Yaskawa INFORM job: SKRZYNIA_5440_-90_STOPNI_20BR.JBI

/JOB
//NAME SKRZYNIA_5440_-90_STOPNI_20BR
///FOLDERNAME 02-SKRZYNIE_JOBS
//POS
///NPOS 563,563,0,37,0,0
///TOOL 0
///POSTYPE PULSE
///PULSE
C00000=0,-52280,40443,0,6876,0
C00001=-82314,-24956,17040,-59626,-27382,-6248
C00002=-93910,-8625,17040,-59626,-43355,-6248
C00003=-98846,-1061,-42166,-80308,-57081,16120
C00004=-100452,6057,-48127,-85711,-56704,21322
C00005=-95817,31791,-34187,-84788,-63710,26674
C00006=-95573,33077,-33257,-84645,-64023,26851
C00007=-94315,33778,-32137,-85160,-63467,26714
C00008=-95573,33077,-33257,-84645,-64023,26851
C00009=-94948,31301,-36075,-85235,-63717,27152
C00010=-95573,33077,-33257,-84645,-64023,26851
C00011=-95263,33142,-33256,-84677,-63995,26850
C00012=-95263,33142,-33256,-84677,-63995,26850
C00013=-94230,33719,-32331,-85099,-63538,26735
C00014=-95263,33142,-33256,-84677,-63995,26850
C00015=-94794,31816,-35365,-85120,-63763,27076
C00016=-95263,33142,-33256,-84677,-63995,26850
C00017=-95260,33144,-33256,-84678,-63995,26850
C00018=-95260,33144,-33256,-84678,-63995,26850
C00019=-94260,33701,-32361,-85086,-63552,26738
C00020=-95260,33144,-33256,-84678,-63995,26850
C00021=-94835,31943,-35167,-85080,-63786,27056
C00022=-95260,33144,-33256,-84678,-63995,26850
C00023=-95258,25631,32269,-66559,-75499,2416
C00024=-95258,25631,32269,-66559,-75499,2416
C00025=-94256,26435,33444,-66420,-74940,2208
C00026=-95258,25631,32269,-66559,-75499,2416
C00027=-94857,24030,29962,-66606,-75105,2539
C00028=-95258,25631,32269,-66559,-75499,2416
C00029=-98811,21047,-15512,-99242,-81394,20987
C00030=-98811,21047,-15512,-99242,-81394,20987
C00031=-97856,21592,-14760,-99539,-80803,20995
C00032=-98811,21047,-15512,-99242,-81394,20987
C00033=-98487,19855,-17143,-99373,-81250,21110
C00034=-98811,21047,-15512,-99242,-81394,20987
C00035=-99077,36985,67047,-90824,-74996,11
C00036=-99077,36985,67047,-90824,-74996,11
C00037=-98126,38026,68808,-90519,-74354,-175
C00038=-99077,36985,67047,-90824,-74996,11
C00039=-98675,34279,62554,-90994,-74807,523
C00040=-99077,36985,67047,-90824,-74996,11
C00041=-98046,30065,45001,-99674,-75008,5996
C00042=-96663,27244,32711,-106417,-76052,10001
C00043=-96035,27733,33435,-106407,-75606,10011
C00044=-96663,27244,32711,-106417,-76052,10001
C00045=-96274,25568,30264,-106516,-75947,10234
C00046=-96663,27244,32711,-106417,-76052,10001
C00047=-93416,-2088,4699,-99676,-50441,9343
C00048=-88080,-20128,-3199,-80943,-31244,2335
C00049=-48287,-55439,-44481,-48508,-5390,-10469
C00050=-48287,-44591,-17414,-16172,-14532,-25809
C00051=-73855,-32171,-5678,-43952,-33220,-11069
C00052=-84843,-2315,38096,-46044,-43440,-11681
C00053=-99590,25338,21334,-81459,-78469,-3358
C00054=-99590,25338,21334,-81459,-78469,-3358
C00055=-98681,25943,22203,-81468,-77867,-3455
C00056=-99590,25338,21334,-81459,-78469,-3358
C00057=-99296,24016,19444,-81525,-78239,-3225
C00058=-99590,25338,21334,-81459,-78469,-3358
C00059=-99820,26032,21623,-82067,-78848,-4447
C00060=-99820,26032,21623,-82067,-78848,-4447
C00061=-98898,26645,22513,-82083,-78237,-4546
C00062=-99820,26032,21623,-82067,-78848,-4447
C00063=-99438,24292,19129,-82156,-78552,-4268
C00064=-99820,26032,21623,-82067,-78848,-4447
C00065=-95331,1432,-9864,-84798,-60031,-3557
C00066=-91210,-11403,-27677,-113165,-52408,5733
C00067=-98271,-15326,-41207,-114268,-59488,7673
C00068=-83743,-25164,-57719,-138536,-50905,17366
C00069=-83743,-25361,-52011,-136459,-47698,15842
C00070=-93071,-30029,-62286,-132724,-54351,14554
C00071=-61872,-66272,-83954,-148251,-32298,21081
C00072=-61872,-49557,-32264,-110357,-15428,1928
C00073=-65143,-26385,24751,-20080,-56896,-30933
C00074=-90244,4395,51028,-38516,-59607,-23032
C00075=-79356,-9150,9683,-42499,-40407,-18801
C00076=-98951,25836,42573,-74290,-75705,-4216
C00077=-99097,30513,38864,-76423,-80199,-875
C00078=-97872,31473,40332,-76298,-79437,-1085
C00079=-99097,30513,38864,-76423,-80199,-875
C00080=-98774,28880,36400,-76469,-79893,-679
C00081=-99097,30513,38864,-76423,-80199,-875
C00082=-99862,24525,29609,-86160,-76987,1407
C00083=-99452,22245,7122,-97683,-80070,9369
C00084=-99292,23987,9562,-97373,-81102,9104
C00085=-98184,24694,10564,-97522,-80343,9095
C00086=-99292,23987,9562,-97373,-81102,9104
C00087=-99030,22873,7999,-97442,-80972,9229
C00088=-99292,23987,9562,-97373,-81102,9104
C00089=-95017,-9844,-333,-79976,-47193,-2364
C00090=-62804,-32782,1918,-36164,-30925,-23493
C00091=-48283,-21883,28214,-25170,-26491,48363
C00092=-45951,-10962,51022,-17493,-32991,44756
C00093=-50347,-18571,12268,-49104,-16423,60029
C00094=-52008,-16476,13921,-52720,-16985,61589
C00095=-50839,-15356,14836,-51561,-16264,61168
C00096=-51137,-15647,14596,-51864,-16447,61279
C00097=-52695,-14846,15261,-54465,-17168,62360
C00098=-51384,-16746,13703,-51673,-16698,61154
C00099=-50347,-18571,12268,-49104,-16423,60029
C00100=-52476,-17044,12146,-55476,-16783,62883
C00101=-51467,-16091,12918,-54586,-16145,62570
C00102=-51762,-16375,12685,-54854,-16332,62665
C00103=-53129,-15664,13268,-57063,-16995,63582
C00104=-52557,-17119,12084,-55547,-16837,62908
C00105=-50509,-19000,10610,-51503,-15997,61182
C00106=-52966,-16930,12240,-56194,-17032,63176
C00107=-51879,-15912,13067,-55265,-16346,62852
C00108=-52154,-16175,12851,-55507,-16521,62938
C00109=-53227,-15612,13314,-57215,-17042,63646
C00110=-52966,-16930,12240,-56194,-17032,63176
C00111=-50703,-18403,11066,-52155,-16024,61477
C00112=-52780,-17619,11680,-55562,-17015,62889
C00113=-51306,-16241,12790,-54268,-16084,62435
C00114=-51660,-16583,12512,-54593,-16308,62551
C00115=-53327,-15718,13220,-57282,-17114,63667
C00116=-52780,-17619,11680,-55562,-17015,62889
C00117=-50704,-18401,11069,-52157,-16021,61478
C00118=-53191,-17342,11901,-56260,-17204,63181
C00119=-51773,-16022,12969,-55050,-16305,62760
C00120=-52146,-16378,12679,-55379,-16540,62876
C00121=-53214,-15820,13135,-57085,-17059,63584
C00122=-53002,-17172,12037,-56105,-17083,63128
C00123=-51005,-17995,11387,-52847,-16122,61778
C00124=-52654,-17319,11922,-55560,-16911,62904
C00125=-51372,-16113,12897,-54432,-16099,62508
C00126=-51648,-16379,12679,-54684,-16273,62598
C00127=-52952,-15703,13233,-56807,-16903,63480
C00128=-53323,-17134,12070,-56539,-17248,63304
C00129=-52826,-20105,4812,-63938,-15678,66983
C00130=-52298,-19620,5183,-63681,-15322,66914
C00131=-51076,-18450,6096,-63049,-14499,66733
C00132=-51419,-18785,5831,-63233,-14731,66786
C00133=-52680,-18133,6347,-65138,-15424,67581
C00134=-52924,-19431,7025,-60935,-16175,65505
C00135=-51752,-18759,10786,-53484,-16613,62002
C00136=-52244,-17884,11471,-54682,-16766,62529
C00137=-50303,-16031,12961,-52880,-15542,61887
C00138=-50741,-16464,12607,-53310,-15818,62044
C00139=-52416,-15612,13306,-56135,-16617,63223
C00140=-51898,-18011,11369,-54129,-16600,62301
C00141=-50945,-18019,11363,-52741,-16103,61737
C00142=-51347,-17395,11856,-53690,-16237,62152
C00143=-49990,-16073,12923,-52376,-15383,61677
C00144=-50384,-16465,12603,-52769,-15629,61822
C00145=-52066,-15616,13298,-55654,-16423,63028
C00146=-51792,-17610,11685,-54205,-16494,62350
C00147=-50945,-18019,11363,-52741,-16103,61737
C00148=-50845,-17493,11778,-52895,-15987,61824
C00149=-49521,-16191,12826,-51571,-15155,61341
C00150=-49894,-16567,12520,-51958,-15389,61484
C00151=-51728,-15654,13268,-55171,-16246,62832
C00152=-51082,-17431,11827,-53280,-16102,61986
C00153=-50028,-23690,-6096,-22921,-31075,54538
C00154=-50346,-22995,-5584,-23393,-31002,54768
C00155=-48843,-21430,-4410,-21901,-30270,54078
C00156=-49178,-21788,-4683,-22239,-30433,54235
C00157=-50538,-21100,-4158,-23908,-30654,55032
C00158=-50252,-22811,-5450,-23315,-30936,54734
C00159=-49763,-24818,-32918,-23163,-28604,59699
C00160=-49144,-24298,-32242,-22455,-28505,59304
C00161=-47766,-22458,-30816,-21237,-27774,58615
C00162=-48099,-22913,-31171,-21534,-27949,58786
C00163=-49602,-21997,-30448,-23301,-28174,59772
C00164=-49259,-23869,-32392,-22880,-28141,59533
C00165=-50713,-12366,-58367,-41124,-17813,74400
C00166=-50097,-11438,-57505,-40749,-17495,74109
C00167=-49105,-9842,-55994,-40096,-16991,73614
C00168=-49355,-10250,-56383,-40269,-17116,73742
C00169=-50506,-9357,-55529,-41571,-17503,74586
C00170=-49771,-10920,-57018,-40545,-17327,73951
C00171=-46548,-30139,-39639,-20061,-27197,57955
C00172=-48797,-26670,-6576,-20404,-32539,53259
C00173=-45389,-28224,4312,-35967,-15579,54278
C00174=-40154,-51179,-915,-24203,-8234,36524
C00175=0,-52280,40443,0,6876,0
C00176=-2117,-50103,-33543,-4117,45077,85249
C00177=26439,-48928,-33543,-4117,-52362,85249
C00178=26439,-27355,-33543,-41485,-52362,85249
C00179=39218,-24492,-41653,-51934,-39374,86964
C00180=38244,-2284,-24157,-56964,-37300,90090
C00181=26640,586,-20198,-77712,-51919,89712
C00182=26323,460,-20341,-77681,-52125,89737
C00183=25607,3186,-17293,-77585,-52601,89760
C00184=26323,460,-20341,-77681,-52125,89737
C00185=27719,1044,-19697,-77798,-51218,89644
C00186=26640,586,-20198,-77712,-51919,89712
C00187=46457,7101,-11330,-26648,-40775,82885
C00188=47439,8350,-9833,-26106,-40556,82449
C00189=46334,10684,-6981,-26557,-41070,82837
C00190=47439,8350,-9833,-26106,-40556,82449
C00191=48354,9159,-8854,-25603,-40343,82046
C00192=47439,8350,-9833,-26106,-40556,82449
C00193=24760,-3019,-10726,-94610,-54398,89614
C00194=25145,-1220,-8811,-94681,-54143,89655
C00195=24492,1290,-6066,-94601,-54582,89624
C00196=25145,-1220,-8811,-94681,-54143,89655
C00197=26584,-669,-8211,-94866,-53174,89734
C00198=25145,-1220,-8811,-94681,-54143,89655
C00199=14532,-15164,-22494,-92943,-61192,88617
C00200=-33377,-12679,-20251,-90012,-93751,87621
C00201=-32674,-7309,22058,-70557,-98373,80594
C00202=20046,-29908,-41690,-58842,-55822,75080
C00203=46158,10269,-6164,-23128,-46470,70172
C00204=51306,10256,-19432,-23475,-33025,71236
C00205=50386,12004,-17260,-23922,-33430,71616
C00206=51306,10256,-19432,-23475,-33025,71236
C00207=51995,10928,-18601,-23012,-32906,70879
C00208=51306,10256,-19432,-23475,-33025,71236
C00209=50667,8104,-22050,-23976,-33027,71608
C00210=27434,3323,14960,-56922,-57501,78346
C00211=29014,6574,18756,-56344,-56678,77965
C00212=28326,9009,21700,-56459,-57175,78009
C00213=29014,6574,18756,-56344,-56678,77965
C00214=30292,7183,19486,-55908,-55969,77693
C00215=29014,6574,18756,-56344,-56678,77965
C00216=24457,-1296,-8898,-94600,-54606,89622
C00217=24457,-1296,-8898,-94600,-54606,89622
C00218=23939,748,-6672,-94541,-54956,89598
C00219=24457,-1296,-8898,-94600,-54606,89622
C00220=25626,-864,-8432,-94748,-53818,89684
C00221=24457,-1296,-8898,-94600,-54606,89622
C00222=22058,-20035,-26567,-93333,-56013,88551
C00223=-28907,-25632,-31027,-90338,-90583,86609
C00224=-23923,-11573,-19230,-90501,-87328,87840
C00225=-8646,-8251,-7782,-76032,-82054,83740
C00226=42001,26537,64712,-25019,-74648,68382
C00227=42692,25604,59505,-25067,-71864,68798
C00228=42100,27723,62792,-25233,-72628,68820
C00229=42692,25604,59505,-25067,-71864,68798
C00230=43179,26157,60355,-24838,-71882,68629
C00231=42692,25604,59505,-25067,-71864,68798
C00232=42064,17796,48100,-25604,-70267,69397
C00233=28113,-7386,-15136,-95790,-47335,90009
C00234=28228,-6488,-14240,-95859,-47266,90053
C00235=27767,-5044,-12775,-95858,-47588,90072
C00236=28228,-6488,-14240,-95859,-47266,90053
C00237=29468,-5989,-13737,-96077,-46438,90154
C00238=28228,-6488,-14240,-95859,-47266,90053
C00239=51937,664,-7429,-160484,-50080,89770
C00240=52345,1107,-6938,-160727,-50007,89930
C00241=51359,2767,-5080,-160136,-50147,89540
C00242=52345,1107,-6938,-160727,-50007,89930
C00243=53054,1752,-6222,-161147,-49882,90209
C00244=52345,1107,-6938,-160727,-50007,89930
C00245=51937,664,-7429,-160484,-50080,89770
C00246=29691,-10745,-18393,-95770,-46230,89933
C00247=26663,-19279,-25970,-94307,-48104,89008
C00248=29542,-7588,-14846,-100915,-46930,90773
C00249=29616,-6902,-10165,-96183,-45225,84004
C00250=29097,-5391,-8640,-96201,-45588,84023
C00251=29616,-6902,-10165,-96183,-45225,84004
C00252=31098,-6282,-9543,-96410,-44233,84135
C00253=29616,-6902,-10165,-96183,-45225,84004
C00254=7576,-30273,-44451,-97512,-61182,86443
C00255=-18624,-40022,-50597,-93591,-78329,83668
C00256=-32134,-30783,-37092,-96173,-88064,83581
C00257=23774,-1324,-8929,-94512,-55065,89585
C00258=23774,-1324,-8929,-94512,-55065,89585
C00259=23319,517,-6924,-94461,-55372,89567
C00260=23774,-1324,-8929,-94512,-55065,89585
C00261=25077,-853,-8421,-94674,-54188,89653
C00262=23774,-1324,-8929,-94512,-55065,89585
C00263=22107,-1052,28039,-94807,-51389,77849
C00264=19995,-16885,24938,-75612,-39910,62837
C00265=8393,-42921,36369,-24238,-5473,19544
C00266=0,-52280,40443,0,6876,0
C00267=-82314,-24956,17040,-59626,-27382,-6248
C00268=-93910,-8625,17040,-59626,-43355,-6248
C00269=-98846,-1061,-42166,-80308,-57081,16120
C00270=-100452,6057,-48127,-85711,-56704,21322
C00271=-95564,34698,-34234,-85516,-63941,27819
C00272=-94021,36658,-30981,-84167,-64832,27454
C00273=-93851,36773,-30815,-84181,-64812,27439
C00274=-95564,34698,-34234,-85516,-63941,27819
C00275=-96930,32282,-32252,-82595,-65816,26305
C00276=-93901,32995,-31122,-83953,-64436,26132
C00277=-93891,32978,-31150,-83961,-64431,26134
C00278=-96930,32282,-32252,-82595,-65816,26305
C00279=-97719,-4194,-31542,-76086,-54596,10626
C00280=-88377,-34186,-45291,-67238,-52212,2442
C00281=-73560,-62084,7826,-28695,-34737,-3666
C00282=0,-52280,40443,0,6876,0
C00283=0,-52280,40443,0,6876,0
C00284=-2117,-50103,-33543,-4117,45077,85249
C00285=26439,-48928,-33543,-4117,-52362,85249
C00286=26439,-27355,-33543,-41485,-52362,85249
C00287=39218,-24492,-41653,-51934,-39374,86964
C00288=37381,-5106,-22608,-53943,-39515,88347
C00289=38119,-10689,-19379,-70548,-34101,88029
C00290=37906,-14512,-22901,-69984,-34376,87713
C00291=41414,6981,-5927,-33889,-45598,86373
C00292=42289,10624,-1511,-33365,-45508,85956
C00293=42351,10656,-1473,-33340,-45486,85935
C00294=41414,6981,-5927,-33889,-45598,86373
C00295=53221,-12364,-8957,-19277,-47766,73858
C00296=11365,-15171,10010,-30164,-77975,82960
C00297=16156,-38280,11293,-23671,-42998,42040
C00298=11365,-47379,10010,-30164,3063,681
C00299=0,-52280,40443,0,6876,0
C00300=0,-36700,24612,42871,-31823,33862
C00301=-44403,-30110,7154,-24155,-23805,45557
C00302=-51570,-19542,10947,-41619,-21811,53396
C00303=-51570,-17239,16856,-38066,-23574,51584
C00304=-55052,-13712,19754,-43494,-24529,53873
C00305=-55190,-12778,21730,-42693,-25060,53437
C00306=-40431,-28773,9158,-17648,-23273,42875
C00307=0,-36700,24612,42871,-31823,33862
C00308=0,-52280,40443,0,6876,0
C00309=0,-52280,40443,0,6876,0
C00310=-73560,-62084,7826,-28695,-34737,-3666
C00311=-88377,-34186,-45291,-67238,-52212,2442
C00312=-99860,-8392,-35780,-75647,-56000,10650
C00313=-100432,21324,12575,-83706,-77956,7498
C00314=-100432,21324,12575,-83706,-77956,7498
C00315=-97477,24790,17443,-83584,-77881,7143
C00316=-97548,25214,18044,-83537,-78171,7107
C00317=-100432,21324,12575,-83706,-77956,7498
C00318=-100473,21504,12824,-83696,-77986,7482
C00319=-97708,25565,18549,-83502,-78342,7077
C00320=-97720,26100,19317,-83456,-78605,7025
C00321=-100432,21324,12575,-83706,-77956,7498
C00322=-98403,3681,-8965,-86029,-63956,7946
C00323=-98851,2841,7216,-80537,-62817,1838
C00324=-99868,-33,22146,-72719,-59601,-5126
C00325=-99028,-10516,17309,-71061,-60695,-4227
C00326=-58820,-39124,10926,-53325,-41870,-3759
C00327=0,-52280,40443,0,6876,0
C00328=-37281,-50778,-9546,-79570,-75313,71156
C00329=-21038,-23698,-30323,-82948,-81132,85647
C00330=-21230,-24252,-33397,-84866,-81311,86227
C00331=26224,-11477,-22521,-89106,-49066,87170
C00332=30473,789,4724,-68168,-47848,79016
C00333=30460,-1091,-3608,-71823,-46530,81583
C00334=26224,-11477,-22521,-89106,-49066,87170
C00335=1250,-26379,-34995,-85812,-66036,85728
C00336=-29373,-17697,-13794,-84248,-87305,82376
C00337=-12562,-22815,-22029,-52123,-75138,85349
C00338=41964,2536,-13642,-34848,-42769,74522
C00339=37974,4101,-26304,-58477,-36842,84551
C00340=37992,4823,-31618,-63468,-34913,87461
C00341=41439,5489,-14791,-37032,-40569,75962
C00342=38833,-3286,10682,-41231,-51577,69207
C00343=-9276,-22918,-17698,-90837,-69000,78700
C00344=-8172,-56778,-49528,-75726,-40055,75711
C00345=-3982,-61001,-53003,-69042,-33087,73336
C00346=37287,-55159,35520,-2191,5667,2084
C00347=0,-52280,40443,0,6876,0
C00348=0,-36700,24612,42871,-31823,33862
C00349=-44403,-30110,7154,-24155,-23805,45557
C00350=-44403,-30110,7154,-24155,-23805,45557
C00351=-42101,-12213,25656,-103795,-5192,78630
C00352=-46259,-8171,27719,-110365,-8144,81138
C00353=-67532,2461,52564,-58221,-38014,54436
C00354=-67092,2390,52438,-57975,-37749,54380
C00355=-61198,-4613,8805,-137219,-40022,88160
C00356=-56934,-15752,2926,-132390,-27589,90381
C00357=-47073,-34549,9488,-27883,-30316,51458
C00358=0,-52280,40443,0,6876,0
C00359=0,-52280,40443,0,6876,0
C00360=-73560,-62084,7826,-28695,-34737,-3666
C00361=-96366,-17217,16860,-56620,-71703,-18245
C00362=-98152,-14905,2044,-65675,-67485,-3494
C00363=-100467,-7393,-15195,-81625,-60158,6002
C00364=-99336,18440,8642,-84276,-74234,7647
C00365=-99336,18440,8642,-84276,-74234,7647
C00366=-97907,25479,18429,-83510,-78268,7080
C00367=-97774,25771,18838,-83486,-78362,7054
C00368=-99336,18440,8642,-84276,-74234,7647
C00369=-99336,20364,19482,-82786,-74642,4774
C00370=-98337,25059,18813,-87846,-78771,10707
C00371=-98337,23926,10585,-88652,-78855,12971
C00372=-99528,19847,13673,-83665,-74506,6500
C00373=-89817,-17341,-38408,-97132,-45323,12250
C00374=-100347,-21961,-42251,-93939,-52125,11121
C00375=-60204,-59872,-73451,-117647,-17639,18840
C00376=-37721,-67612,11381,-1325,-438,-7850
C00377=0,-52280,40443,0,6876,0
C00378=37287,-55159,35520,-2191,5667,2084
C00379=40042,-68802,-18337,-47708,-19461,45384
C00380=16481,-63411,-38742,-86271,-37962,67106
C00381=28646,-23138,-32952,-89786,-42552,85395
C00382=38882,-16596,-17625,-44304,-41043,72768
C00383=40930,-6862,-13364,-47045,-37020,74415
C00384=41744,-3361,-9781,-46774,-36492,74231
C00385=41678,-4243,-16493,-50979,-33997,76666
C00386=40930,-6862,-13364,-47045,-37020,74415
C00387=38882,-16596,-17625,-44304,-41043,72768
C00388=28646,-23138,-32952,-89786,-42552,85395
C00389=29905,-15291,-26411,-91102,-43435,86304
C00390=31540,-7654,-19248,-92177,-42391,86919
C00391=31445,-8095,-22888,-97196,-43117,89457
C00392=29637,-16450,-35189,-96198,-44206,89682
C00393=-7164,-46429,-55577,-86274,-68578,84143
C00394=40042,-68802,-18337,-47708,-19461,45384
C00395=37287,-55159,35520,-2191,5667,2084
C00396=0,-52280,40443,0,6876,0
C00397=-37164,-60659,6466,-13301,-5027,19773
C00398=-45362,-39990,2831,-27538,-17767,40935
C00399=-57189,-26834,-7130,-38780,-31731,51561
C00400=-55974,-20661,-3180,-39617,-29741,52134
C00401=-55991,-28453,-45977,-64163,-20900,63765
C00402=-57189,-26834,-7130,-38780,-31731,51561
C00403=-41180,-61187,4729,-17280,-8498,23442
C00404=0,-52280,40443,0,6876,0
C00405=0,-52280,40443,0,6876,0
C00406=-43180,-50572,-20637,-6552,-29302,-38834
C00407=-79425,-37128,-15462,-51820,-35721,-18807
C00408=-93702,-21743,-5664,-65079,-41536,-12324
C00409=-94876,-11469,-23586,-124528,-59237,5423
C00410=-92861,23404,17376,-116518,-76732,-1573
C00411=-96665,29896,42633,-98437,-75635,-11031
C00412=-96665,37701,65506,-96077,-73868,-15674
C00413=-98256,26642,30161,-104402,-77650,-7294
C00414=-94876,-11469,-23586,-124528,-59237,5423
C00415=-94108,-26192,-19530,-80749,-38523,-6311
C00416=-79425,-37128,-15462,-51820,-35721,-18807
C00417=-44920,-50063,-20090,-8739,-29356,-37564
C00418=-37721,-67612,11381,-1325,-438,-7850
C00419=0,-52280,40443,0,6876,0
C00420=40043,-68802,-18337,-47706,-19461,45383
C00421=27078,-46675,7729,-35821,-60236,53359
C00422=37661,6027,34279,-36092,-58837,68690
C00423=38848,9668,32452,-36978,-55195,69693
C00424=45203,15557,41040,-24527,-60177,66840
C00425=37661,2340,23735,-37788,-55306,70200
C00426=22173,-30639,7984,-58136,-45615,60133
C00427=37287,-55159,35520,-2191,5667,2084
C00428=0,-52280,40443,0,6876,0
C00429=-23708,-46776,23536,-16027,-4787,19738
C00430=-50917,-40459,4132,-34421,-18173,42391
C00431=-54964,-26842,8528,-44141,-23181,52038
C00432=-51719,-20944,8196,-48593,-18539,54728
C00433=-53338,-16066,12564,-52314,-18938,56375
C00434=-53668,-14237,17353,-48629,-20286,54493
C00435=-18010,-41727,-5437,24633,-20435,23511
C00436=-18010,-41727,-5437,24633,-20435,23511
C00437=-43180,-50572,-20637,-6552,-29302,-38834
C00438=-37721,-67612,11381,-1325,-438,-7850
C00439=0,-52280,40443,0,6876,0
C00440=-7830,-25136,17099,-55306,-64068,52084
C00441=34592,-23156,18291,-29932,-45204,43222
C00442=27626,-5609,7480,-74303,-46810,69713
C00443=30162,-7263,-3756,-79871,-43922,73611
C00444=30945,-3557,12,-79972,-43367,73694
C00445=30934,-3652,-86,-79966,-43372,73693
C00446=29106,-7674,-4162,-79972,-44640,73655
C00447=-2837,-32019,-23857,-80741,-66785,72567
C00448=9534,-43450,13514,-26959,-29486,38723
C00449=22834,-59963,22946,-6692,-2150,9612
C00450=0,-52280,40443,0,6876,0
C00451=-23708,-46776,23536,-16027,-4787,19738
C00452=-50917,-40459,4132,-34421,-18173,42391
C00453=-51059,-36587,4608,-36647,-19418,45358
C00454=-50113,-22729,10834,-36393,-23396,50963
C00455=-58003,-17258,7975,-66354,-22196,69294
C00456=-57660,-15851,11780,-61832,-22634,66694
C00457=-50113,-22729,10834,-36393,-23396,50963
C00458=-45969,-44671,-42317,80322,10570,10889
C00459=-31285,-69981,-10849,-7246,-6842,20992
C00460=0,-52280,40443,0,6876,0
C00461=-37721,-67612,11381,-1325,-438,-7850
C00462=-43180,-50572,-20637,-6552,-29302,-38834
C00463=-92181,-6909,34626,-50562,-49190,-21840
C00464=-101117,-5694,-18308,-85789,-60825,2377
C00465=-97622,-3602,-16155,-86160,-58465,2400
C00466=-99754,24347,18348,-83049,-78046,1543
C00467=-98401,23935,17754,-83131,-77323,1564
C00468=-98274,24050,17917,-83129,-77329,1551
C00469=-99954,24418,19993,-82828,-78557,1051
C00470=-99712,24798,18984,-83012,-78332,1506
C00471=-99852,25442,19906,-82977,-78439,1439
C00472=-98294,26390,21274,-82926,-78604,1336
C00473=-98320,27540,23370,-82787,-79202,1083
C00474=-99852,25442,19906,-82977,-78439,1439
C00475=-99768,8894,-2445,-89351,-68751,3793
C00476=-96099,-3787,-16815,-92200,-58195,4535
C00477=-97559,-25159,-36085,-93407,-46496,3918
C00478=-68601,-52593,-52127,-95725,-25602,3235
C00479=-80632,-38079,-20908,-64053,-45216,-12949
C00480=-43180,-50572,-20637,-6552,-29302,-38834
C00481=-37721,-67612,11381,-1325,-438,-7850
C00482=54026,-30203,28811,7745,-28969,5087
C00483=55906,-29650,27841,6704,-28568,42061
C00484=3910,-49110,-20873,-64325,-51391,71742
C00485=9596,-41005,-15480,-61992,-50741,70573
C00486=34629,-5327,8260,-51720,-47880,65426
C00487=35679,2837,17551,-51053,-47466,65038
C00488=35689,-56,7549,-54586,-44718,67469
C00489=34629,-5327,8260,-51720,-47880,65426
C00490=9596,-41005,-15480,-61992,-50741,70573
C00491=29660,-4584,-26917,-122917,-59269,85605
C00492=30458,-1431,-23593,-123278,-58903,85810
C00493=32051,-581,-21149,-126899,-58917,85995
C00494=28378,-5181,-30467,-124970,-61925,86269
C00495=9596,-41005,-15480,-61992,-50741,70573
C00496=4124,-42500,-16101,-63937,-54198,71061
C00497=22834,-59963,22946,-6692,-2150,9612
C00498=0,-52280,40443,0,6876,0
C00499=-44101,-76445,-48847,-15697,-17168,40457
C00500=-48984,-30078,-36716,-21434,-29637,58750
C00501=-50484,-13386,-55713,-36158,-19724,71897
C00502=-50319,-9878,-52358,-36554,-19395,72071
C00503=-57778,15231,-57159,-77377,-21293,89265
C00504=-57778,15231,-57159,-77377,-21293,89265
C00505=-50484,-13386,-55713,-36158,-19724,71897
C00506=-49763,-25421,-36239,-24565,-26935,60445
C00507=-50529,-22709,-3778,-22940,-31995,54502
C00508=-45389,-28224,4312,-35967,-15579,54278
C00509=-40154,-51179,-915,-24203,-8234,36524
C00510=0,-52280,40443,0,6876,0
C00511=0,-52280,40443,0,6876,0
C00512=-37721,-67612,11381,-1325,-438,-7850
C00513=-43180,-50572,-20637,-6552,-29302,-38834
C00514=-43180,-50572,-20637,-6552,-29302,-38834
C00515=-91233,-13472,9135,-57436,-42793,-15671
C00516=-94453,18451,26397,-64403,-69695,-4898
C00517=-94848,25710,19994,-67599,-74328,1083
C00518=-94734,25454,19627,-67614,-74234,1097
C00519=-94605,24228,10738,-68938,-72404,3439
C00520=-96555,21614,11724,-68276,-72695,2131
C00521=-99000,22482,23037,-75261,-76004,639
C00522=-97210,28604,31066,-74659,-78513,378
C00523=-97154,26647,21384,-75593,-77346,2770
C00524=-100531,16612,13557,-75306,-72509,1088
C00525=-98914,15791,22093,-91892,-69242,2220
C00526=-98524,31242,37673,-92432,-80087,2200
C00527=-98508,35203,51300,-91477,-79539,-794
C00528=-99299,29399,42249,-91532,-77608,155
C00529=-99299,39874,71997,-89061,-76925,-5800
C00530=-98153,38420,66100,-91432,-76531,-4068
C00531=-98147,36464,60868,-91873,-76694,-3060
C00532=-99718,12303,6039,-96207,-71156,6635
C00533=-93032,-8711,-3060,-81304,-48072,-4095
C00534=-98228,-14972,-11291,-81392,-49231,-4002
C00535=-91129,-17870,8831,-66292,-48444,-14183
C00536=-68865,-35989,-5252,-49829,-38105,-21179
C00537=-15566,-52364,-9989,12732,-35649,-46896
C00538=0,-52278,40443,-31822,-65283,46097
C00539=7820,3000,44222,-77356,-66876,70486
C00540=23103,22769,71034,-65639,-61603,67373
C00541=25078,30713,84198,-63240,-61811,65668
C00542=25008,30264,83410,-63369,-61766,65773
C00543=23103,22769,71034,-65639,-61603,67373
C00544=23103,22769,71034,-65639,-61603,67373
C00545=25078,30713,84198,-63240,-61811,65668
C00546=25008,30264,83410,-63369,-61766,65773
C00547=23103,22769,71034,-65639,-61603,67373
C00548=-3014,-20441,-7349,-104591,-68614,79454
C00549=-3014,-20441,-7349,-104591,-68614,79454
C00550=-13238,-21720,-1359,-93359,-59492,72612
C00551=10261,-46634,14475,-36899,-22136,31570
C00552=22834,-59963,22946,-6692,-2150,9612
C00553=0,-52280,40443,0,6876,0
C00554=-23708,-46776,23536,-16027,-4787,19738
C00555=-50917,-40459,4132,-34421,-18173,42391
C00556=-49876,-21948,7530,-68838,-10324,59148
C00557=-46721,-18942,9765,-68167,-8197,59205
C00558=-47734,-15041,12007,-78406,-8476,63945
C00559=-48173,-14749,12492,-78097,-8776,63748
C00560=-42573,-24036,4541,-56448,-5917,54155
C00561=-31287,-69981,-10850,-7253,-6843,20996
C00562=0,-52280,40443,0,6876,0
BC00000=455888
BC00001=445130
BC00002=445130
BC00003=445130
BC00004=445130
BC00005=467179
BC00006=468227
BC00007=468227
BC00008=468227
BC00009=468227
BC00010=468227
BC00011=514421
BC00012=514421
BC00013=514421
BC00014=514421
BC00015=514421
BC00016=514421
BC00017=560588
BC00018=560588
BC00019=560588
BC00020=560588
BC00021=560588
BC00022=560588
BC00023=536404
BC00024=536404
BC00025=536404
BC00026=536404
BC00027=536404
BC00028=536404
BC00029=582458
BC00030=582458
BC00031=582458
BC00032=582458
BC00033=582458
BC00034=582458
BC00035=581206
BC00036=581206
BC00037=581206
BC00038=581206
BC00039=581206
BC00040=581206
BC00041=608443
BC00042=626741
BC00043=626741
BC00044=626741
BC00045=626741
BC00046=626741
BC00047=604255
BC00048=604255
BC00049=627238
BC00050=699121
BC00051=730161
BC00052=730161
BC00053=820815
BC00054=820815
BC00055=820815
BC00056=820815
BC00057=820815
BC00058=820815
BC00059=866263
BC00060=866263
BC00061=866263
BC00062=866263
BC00063=866263
BC00064=866263
BC00065=866263
BC00066=872244
BC00067=872244
BC00068=872244
BC00069=872244
BC00070=872244
BC00071=872244
BC00072=872244
BC00073=967932
BC00074=965893
BC00075=970341
BC00076=974685
BC00077=981233
BC00078=981233
BC00079=981233
BC00080=981233
BC00081=981233
BC00082=979269
BC00083=1044956
BC00084=1044956
BC00085=1044956
BC00086=1044956
BC00087=1044956
BC00088=1044956
BC00089=978491
BC00090=968330
BC00091=919701
BC00092=943157
BC00093=1012084
BC00094=1012084
BC00095=1012084
BC00096=1012084
BC00097=1012084
BC00098=1012084
BC00099=949003
BC00100=953382
BC00101=953382
BC00102=953382
BC00103=953382
BC00104=953382
BC00105=888056
BC00106=888056
BC00107=888056
BC00108=888056
BC00109=888056
BC00110=888056
BC00111=830714
BC00112=830714
BC00113=830714
BC00114=830714
BC00115=830714
BC00116=830714
BC00117=764829
BC00118=764829
BC00119=764829
BC00120=764829
BC00121=764829
BC00122=764829
BC00123=707174
BC00124=707174
BC00125=707174
BC00126=707174
BC00127=707174
BC00128=707174
BC00129=642071
BC00130=642071
BC00131=642071
BC00132=642071
BC00133=642071
BC00134=642071
BC00135=584746
BC00136=584746
BC00137=584746
BC00138=584746
BC00139=584746
BC00140=584746
BC00141=519232
BC00142=519232
BC00143=519232
BC00144=519232
BC00145=519232
BC00146=519232
BC00147=461813
BC00148=461813
BC00149=461813
BC00150=461813
BC00151=461813
BC00152=461813
BC00153=459544
BC00154=459544
BC00155=459544
BC00156=459544
BC00157=459544
BC00158=459544
BC00159=459544
BC00160=459544
BC00161=459544
BC00162=459544
BC00163=459544
BC00164=459544
BC00165=459544
BC00166=459544
BC00167=459544
BC00168=459544
BC00169=459544
BC00170=459544
BC00171=459544
BC00172=459544
BC00173=459540
BC00174=533216
BC00175=533216
BC00176=423885
BC00177=423885
BC00178=423885
BC00179=423885
BC00180=423885
BC00181=423882
BC00182=423882
BC00183=423882
BC00184=423882
BC00185=423882
BC00186=423882
BC00187=517447
BC00188=516208
BC00189=516208
BC00190=516208
BC00191=516208
BC00192=516208
BC00193=462401
BC00194=462401
BC00195=462401
BC00196=462401
BC00197=462401
BC00198=462401
BC00199=462401
BC00200=462401
BC00201=581968
BC00202=647467
BC00203=647467
BC00204=647467
BC00205=647467
BC00206=647467
BC00207=647467
BC00208=647467
BC00209=647467
BC00210=600589
BC00211=600589
BC00212=600589
BC00213=600589
BC00214=600589
BC00215=600589
BC00216=646713
BC00217=646713
BC00218=646713
BC00219=646713
BC00220=646713
BC00221=646713
BC00222=646713
BC00223=646713
BC00224=703926
BC00225=764819
BC00226=734650
BC00227=734650
BC00228=734650
BC00229=734650
BC00230=734650
BC00231=734650
BC00232=734650
BC00233=762000
BC00234=762000
BC00235=762000
BC00236=762000
BC00237=762000
BC00238=762000
BC00239=768744
BC00240=768744
BC00241=768744
BC00242=768744
BC00243=768744
BC00244=768744
BC00245=768744
BC00246=762000
BC00247=762000
BC00248=869424
BC00249=869424
BC00250=869424
BC00251=869424
BC00252=869424
BC00253=869424
BC00254=869424
BC00255=869424
BC00256=983898
BC00257=992364
BC00258=992364
BC00259=992364
BC00260=992364
BC00261=992364
BC00262=992364
BC00263=927243
BC00264=910363
BC00265=854316
BC00266=458496
BC00267=445130
BC00268=445130
BC00269=445130
BC00270=445130
BC00271=475938
BC00272=475917
BC00273=468314
BC00274=475938
BC00275=515329
BC00276=515329
BC00277=508301
BC00278=515329
BC00279=542207
BC00280=542207
BC00281=542207
BC00282=542207
BC00283=492150
BC00284=423885
BC00285=423885
BC00286=423885
BC00287=423885
BC00288=418215
BC00289=406365
BC00290=406365
BC00291=507950
BC00292=507950
BC00293=500226
BC00294=507950
BC00295=493160
BC00296=493160
BC00297=493160
BC00298=493160
BC00299=493160
BC00300=582810
BC00301=655182
BC00302=714528
BC00303=712780
BC00304=712780
BC00305=773753
BC00306=773753
BC00307=582810
BC00308=540924
BC00309=542207
BC00310=542207
BC00311=542207
BC00312=590944
BC00313=543764
BC00314=459277
BC00315=459277
BC00316=451665
BC00317=459277
BC00318=520748
BC00319=520748
BC00320=528295
BC00321=520748
BC00322=524597
BC00323=612873
BC00324=584417
BC00325=584417
BC00326=584417
BC00327=584417
BC00328=542360
BC00329=599440
BC00330=482963
BC00331=482963
BC00332=482963
BC00333=482963
BC00334=482963
BC00335=482963
BC00336=482963
BC00337=633179
BC00338=633182
BC00339=633182
BC00340=633182
BC00341=633182
BC00342=590162
BC00343=577838
BC00344=565789
BC00345=612529
BC00346=620193
BC00347=620193
BC00348=812803
BC00349=887783
BC00350=927066
BC00351=893694
BC00352=914884
BC00353=934809
BC00354=991752
BC00355=1014590
BC00356=945981
BC00357=853059
BC00358=542207
BC00359=542207
BC00360=513519
BC00361=556866
BC00362=576802
BC00363=590944
BC00364=571989
BC00365=566860
BC00366=566866
BC00367=572997
BC00368=566860
BC00369=625806
BC00370=632891
BC00371=631419
BC00372=627770
BC00373=635118
BC00374=635118
BC00375=633159
BC00376=733103
BC00377=733103
BC00378=620193
BC00379=620193
BC00380=625652
BC00381=635598
BC00382=635598
BC00383=635598
BC00384=635598
BC00385=635598
BC00386=635598
BC00387=635598
BC00388=635598
BC00389=658627
BC00390=658630
BC00391=665879
BC00392=658627
BC00393=658627
BC00394=620193
BC00395=620193
BC00396=620193
BC00397=561542
BC00398=498768
BC00399=452071
BC00400=452071
BC00401=452071
BC00402=452071
BC00403=524165
BC00404=524165
BC00405=733103
BC00406=733103
BC00407=615417
BC00408=615411
BC00409=615411
BC00410=615411
BC00411=623591
BC00412=623591
BC00413=621042
BC00414=615411
BC00415=615411
BC00416=636921
BC00417=698572
BC00418=733103
BC00419=733103
BC00420=667407
BC00421=721208
BC00422=721208
BC00423=721208
BC00424=727232
BC00425=730010
BC00426=686453
BC00427=620193
BC00428=620193
BC00429=576077
BC00430=541793
BC00431=580754
BC00432=589556
BC00433=589433
BC00434=647350
BC00435=649294
BC00436=769586
BC00437=795297
BC00438=733103
BC00439=733103
BC00440=727492
BC00441=727492
BC00442=759331
BC00443=759331
BC00444=759331
BC00445=766564
BC00446=759331
BC00447=759331
BC00448=672725
BC00449=672725
BC00450=672725
BC00451=766882
BC00452=791101
BC00453=802867
BC00454=836517
BC00455=836517
BC00456=895002
BC00457=836517
BC00458=798026
BC00459=767805
BC00460=733103
BC00461=733103
BC00462=733103
BC00463=733103
BC00464=815675
BC00465=817504
BC00466=817504
BC00467=817504
BC00468=824335
BC00469=824335
BC00470=862603
BC00471=862905
BC00472=863393
BC00473=870426
BC00474=862905
BC00475=824848
BC00476=818776
BC00477=812035
BC00478=750469
BC00479=783373
BC00480=795297
BC00481=733103
BC00482=762701
BC00483=765633
BC00484=830967
BC00485=835024
BC00486=852883
BC00487=852883
BC00488=852883
BC00489=852883
BC00490=835024
BC00491=861491
BC00492=861491
BC00493=861491
BC00494=861491
BC00495=835024
BC00496=835024
BC00497=672725
BC00498=672725
BC00499=528256
BC00500=459544
BC00501=459544
BC00502=459544
BC00503=459544
BC00504=450616
BC00505=459544
BC00506=459544
BC00507=459544
BC00508=459540
BC00509=533216
BC00510=533216
BC00511=733103
BC00512=733103
BC00513=854587
BC00514=971430
BC00515=966378
BC00516=992810
BC00517=992810
BC00518=992810
BC00519=992810
BC00520=992810
BC00521=992810
BC00522=992810
BC00523=992810
BC00524=990650
BC00525=1014865
BC00526=1014865
BC00527=1014865
BC00528=1014865
BC00529=1014865
BC00530=1014865
BC00531=1027264
BC00532=1027264
BC00533=979788
BC00534=976838
BC00535=956699
BC00536=952322
BC00537=952322
BC00538=921533
BC00539=921533
BC00540=946591
BC00541=946591
BC00542=953713
BC00543=946591
BC00544=997282
BC00545=997282
BC00546=1004404
BC00547=997282
BC00548=1013986
BC00549=963295
BC00550=908449
BC00551=754884
BC00552=672725
BC00553=672725
BC00554=562340
BC00555=452362
BC00556=452362
BC00557=452362
BC00558=452362
BC00559=512870
BC00560=511886
BC00561=742282
BC00562=742282
///POSTYPE BASE
///RECTAN
///RCONF 0,0,0,0,0,0,0,0,0,0,0,0,0,0,0,0,0,0,0,0,0,0,0,0
P00006=-2.449,0.031,8.825,0.0000,0.0000,0.0000
///RCONF 1,0,0,0,0,0,0,0,0,0,0,0,0,0,0,0,0,0,0,0,0,0,0,0
P00300=-0.036,-1.505,2.318,0.0000,0.0000,0.0000
///RCONF 0,0,0,0,0,0,0,0,0,0,0,0,0,0,0,0,0,0,0,0,0,0,0,0
P00301=0.005,-4.708,-4.628,0.0000,0.0000,0.0000
P00302=0.052,-2.937,-4.426,0.0000,0.0000,0.0000
P00303=-0.004,-1.437,-4.584,0.0000,0.0000,0.0000
P00304=0.028,-1.666,-4.234,0.0000,0.0000,0.0000
P00305=-0.003,-1.920,-3.501,0.0000,0.0000,0.0000
P00306=0.015,-2.252,-3.054,0.0000,0.0000,0.0000
P00308=-0.003,-2.092,-4.888,0.0000,0.0000,0.0000
P00309=-0.040,-2.205,-4.992,0.0000,0.0000,0.0000
P00311=-0.007,-2.079,-5.307,0.0000,0.0000,0.0000
P00312=-0.032,2.202,-7.632,0.0000,0.0000,0.0000
///RCONF 1,0,0,0,0,0,0,0,0,0,0,0,0,0,0,0,0,0,0,0,0,0,0,0
P00349=0.060,0.167,-1.133,0.0000,0.0000,0.0000
///RCONF 0,0,0,0,0,0,0,0,0,0,0,0,0,0,0,0,0,0,0,0,0,0,0,0
P00350=11.519,-0.008,1.149,0.0000,0.0000,0.0000
P00351=13.563,-0.027,-0.653,0.0000,0.0000,0.0000
P00352=13.252,-0.027,-0.827,0.0000,0.0000,0.0000
P00353=10.971,-0.082,0.776,0.0000,0.0000,0.0000
P00354=-0.024,2.508,-1.824,0.0000,0.0000,0.0000
P00355=-0.001,2.528,-1.131,0.0000,0.0000,0.0000
P00356=-0.034,2.921,-0.262,0.0000,0.0000,0.0000
P00357=0.003,3.386,-0.091,0.0000,0.0000,0.0000
P00358=0.014,3.037,-0.020,0.0000,0.0000,0.0000
P00359=-0.005,2.731,0.912,0.0000,0.0000,0.0000
P00360=-0.011,3.412,0.438,0.0000,0.0000,0.0000
P00361=0.018,3.050,1.253,0.0000,0.0000,0.0000
P00400=5.920,-3.503,-0.024,0.0000,0.0000,0.0000
P00401=3.430,-0.021,1.131,0.0000,0.0000,0.0000
P00402=-0.253,1.107,3.062,0.0000,0.0000,0.0000
P00403=-3.666,-0.015,5.328,0.0000,0.0000,0.0000
///RCONF 1,0,0,0,0,0,0,0,0,0,0,0,0,0,0,0,0,0,0,0,0,0,0,0
P00404=0.029,4.189,-1.030,0.0000,0.0000,0.0000
///RCONF 0,0,0,0,0,0,0,0,0,0,0,0,0,0,0,0,0,0,0,0,0,0,0,0
P00405=2.420,0.007,1.427,0.0000,0.0000,0.0000
P00406=3.513,-0.022,0.429,0.0000,0.0000,0.0000
///RCONF 1,0,0,0,1,0,0,0,0,0,0,0,0,0,0,0,0,0,0,0,0,0,0,0
P00407=-0.029,2.348,-1.469,0.0000,0.0000,0.0000
P00408=0.010,1.346,-1.479,0.0000,0.0000,0.0000
///RCONF 1,0,0,0,0,0,0,0,0,0,0,0,0,0,0,0,0,0,0,0,0,0,0,0
P00409=-0.026,2.090,-1.483,0.0000,0.0000,0.0000
P00410=0.001,4.491,-0.583,0.0000,0.0000,0.0000
///RCONF 1,0,0,0,1,0,0,0,0,0,0,0,0,0,0,0,0,0,0,0,0,0,0,0
P00411=-0.015,3.627,0.872,0.0000,0.0000,0.0000
//INST
///DATE 2024/05/20 13:53
///ATTR SC,RW
///GROUP1 RB1,BS1
NOP
CALL JOB:MOVE_INTO_TUNNEL
MOVJ C00000 BC00000 VJ=30.00
MOVJ C00001 BC00001 VJ=30.00
MOVJ C00002 BC00002 VJ=30.00
MOVL C00003 BC00003 V=500.0
MOVJ C00004 BC00004 VJ=20.00
'------------------------
'W65.3
'------------------------
MOVL C00005 BC00005 V=333.3
MOVL C00006 BC00006 V=166.7 PL=0
REFP 3 C00007 BC00007
CALL JOB:SEARCH-R1
SET P0300 P0006
SFTON P0300
MOVL C00008 BC00008 V=66.7 PL=0
REFP 3 C00009 BC00009
CALL JOB:SEARCH-R1
SET P0300 P0006
SFTON P0300
MOVL C00010 BC00010 V=66.7 PL=0
SFTOF
'------------------------
'W65.5
'------------------------
MOVL C00011 BC00011 V=500.0
MOVL C00012 BC00012 V=166.7 PL=0
REFP 3 C00013 BC00013
CALL JOB:SEARCH-R1
SET P0301 P0006
SFTON P0301
MOVL C00014 BC00014 V=166.7 PL=0
REFP 3 C00015 BC00015
CALL JOB:SEARCH-R1
SET P0301 P0006
SFTON P0301
MOVL C00016 BC00016 V=166.7 PL=0
SFTOF
'------------------------
'W65.7
'------------------------
MOVL C00017 BC00017 V=500.0
MOVL C00018 BC00018 V=166.7 PL=0
REFP 3 C00019 BC00019
CALL JOB:SEARCH-R1
SET P0302 P0006
SFTON P0302
MOVL C00020 BC00020 V=166.7 PL=0
REFP 3 C00021 BC00021
CALL JOB:SEARCH-R1
SET P0302 P0006
SFTON P0302
MOVL C00022 BC00022 V=166.7 PL=0
SFTOF
'------------------------
'W65.10
'------------------------
MOVL C00023 BC00023 V=500.0
MOVL C00024 BC00024 V=166.7 PL=0
REFP 3 C00025 BC00025
CALL JOB:SEARCH-R1
SET P0303 P0006
SFTON P0303
MOVL C00026 BC00026 V=166.7 PL=0
REFP 3 C00027 BC00027
CALL JOB:SEARCH-R1
SET P0303 P0006
SFTON P0303
MOVL C00028 BC00028 V=166.7 PL=0
SFTOF
'------------------------
'W65.12
'------------------------
MOVL C00029 BC00029 V=500.0
MOVL C00030 BC00030 V=166.7 PL=0
REFP 3 C00031 BC00031
CALL JOB:SEARCH-R1
SET P0304 P0006
SFTON P0304
MOVL C00032 BC00032 V=166.7 PL=0
REFP 3 C00033 BC00033
CALL JOB:SEARCH-R1
SET P0304 P0006
SFTON P0304
MOVL C00034 BC00034 V=166.7 PL=0
SFTOF
'------------------------
'W65.15
'------------------------
MOVL C00035 BC00035 V=333.3
MOVL C00036 BC00036 V=166.7 PL=0
REFP 3 C00037 BC00037
CALL JOB:SEARCH-R1
SET P0305 P0006
SFTON P0305
MOVL C00038 BC00038 V=166.7 PL=0
REFP 3 C00039 BC00039
CALL JOB:SEARCH-R1
SET P0305 P0006
SFTON P0305
MOVL C00040 BC00040 V=166.7 PL=0
SFTOF
'------------------------
'W65.17
'------------------------
MOVL C00041 BC00041 V=333.3
MOVL C00042 BC00042 V=166.7 PL=0
REFP 3 C00043 BC00043
CALL JOB:SEARCH-R1
SET P0306 P0006
SFTON P0306
MOVL C00044 BC00044 V=166.7 PL=0
REFP 3 C00045 BC00045
CALL JOB:SEARCH-R1
SET P0306 P0006
SFTON P0306
MOVL C00046 BC00046 V=166.7 PL=0
SFTOF
MOVL C00047 BC00047 V=333.3
MOVL C00048 BC00048 V=500.0
MOVL C00049 BC00049 V=500.0
MOVJ C00050 BC00050 VJ=50.00
MOVL C00051 BC00051 V=500.0
MOVL C00052 BC00052 V=500.0
'------------------------
'W65.20
'------------------------
'------------------------
MOVL C00053 BC00053 V=333.3
MOVL C00054 BC00054 V=166.7 PL=0
REFP 3 C00055 BC00055
CALL JOB:SEARCH-R1
SET P0308 P0006
SFTON P0308
MOVL C00056 BC00056 V=166.7 PL=0
REFP 3 C00057 BC00057
CALL JOB:SEARCH-R1
SET P0308 P0006
SFTON P0308
MOVL C00058 BC00058 V=166.7 PL=0
SFTOF
'------------------------
'W65.25
'------------------------
MOVL C00059 BC00059 V=500.0
MOVL C00060 BC00060 V=166.7 PL=0
REFP 3 C00061 BC00061
CALL JOB:SEARCH-R1
SET P0309 P0006
SFTON P0309
MOVL C00062 BC00062 V=166.7 PL=0
REFP 3 C00063 BC00063
CALL JOB:SEARCH-R1
SET P0309 P0006
SFTON P0309
MOVL C00064 BC00064 V=166.7 PL=0
SFTOF
MOVL C00065 BC00065 V=166.7
MOVL C00066 BC00066 V=666.7
MOVL C00067 BC00067 V=666.7
MOVL C00068 BC00068 V=666.7
MOVL C00069 BC00069 V=666.7
MOVL C00070 BC00070 V=666.7
MOVL C00071 BC00071 V=666.7
MOVL C00072 BC00072 V=666.7
MOVL C00073 BC00073 V=666.7
MOVL C00074 BC00074 V=666.7
MOVL C00075 BC00075 V=666.7
'------------------------
'W65.28
'------------------------
'W65.30
'------------------------
MOVL C00076 BC00076 V=500.0
MOVL C00077 BC00077 V=166.7 PL=0
REFP 3 C00078 BC00078
CALL JOB:SEARCH-R1
SET P0311 P0006
SFTON P0311
MOVL C00079 BC00079 V=166.7 PL=0
REFP 3 C00080 BC00080
CALL JOB:SEARCH-R1
SET P0311 P0006
SFTON P0311
MOVL C00081 BC00081 V=166.7 PL=0
SFTOF
MOVL C00082 BC00082 V=333.3
MOVL C00083 BC00083 V=333.3
MOVL C00084 BC00084 V=166.7
REFP 3 C00085 BC00085
CALL JOB:SEARCH-R1
SET P0312 P0006
SFTON P0312
MOVL C00086 BC00086 V=166.7 PL=0
REFP 3 C00087 BC00087
CALL JOB:SEARCH-R1
SET P0312 P0006
SFTON P0312
MOVL C00088 BC00088 V=166.7 PL=0
SFTOF
MOVL C00089 BC00089 V=333.3
MOVL C00090 BC00090 V=333.3
MOVJ C00091 BC00091 VJ=30.00
MOVJ C00092 BC00092 VJ=30.00
MOVL C00093 BC00093 V=500.0
SFTOF
MOVL C00094 BC00094 V=166.7 PL=0
REFP 3 C00095 BC00095
CALL JOB:SEARCH-R1
SET P0349 P0006
SFTON P0349
MOVL C00096 BC00096 V=166.7 PL=0
REFP 3 C00097 BC00097
CALL JOB:SEARCH-R1
SET P0349 P0006
SFTON P0349
MOVL C00098 BC00098 V=166.7 PL=0
SFTOF
MOVL C00099 BC00099 V=333.3
SFTOF
'------------------------
'W251A
'------------------------
MOVL C00100 BC00100 V=166.7 PL=0
REFP 3 C00101 BC00101
CALL JOB:SEARCH-R1
SET P0350 P0006
SFTON P0350
MOVL C00102 BC00102 V=166.7 PL=0
REFP 3 C00103 BC00103
CALL JOB:SEARCH-R1
SET P0350 P0006
SFTON P0350
MOVL C00104 BC00104 V=166.7 PL=0
SFTOF
'------------------------
'W254A P
'------------------------
MOVJ C00105 BC00105 VJ=40.00
MOVL C00106 BC00106 V=166.7 PL=0
REFP 3 C00107 BC00107
CALL JOB:SEARCH-R1
SET P0351 P0006
SFTON P0351
MOVL C00108 BC00108 V=166.7 PL=0
REFP 3 C00109 BC00109
CALL JOB:SEARCH-R1
SET P0351 P0006
SFTON P0351
MOVL C00110 BC00110 V=166.7 PL=0
SFTOF
'------------------------
'W254A L
'------------------------
MOVJ C00111 BC00111 VJ=40.00
MOVL C00112 BC00112 V=166.7 PL=0
REFP 3 C00113 BC00113
CALL JOB:SEARCH-R1
SET P0352 P0006
SFTON P0352
MOVL C00114 BC00114 V=166.7 PL=0
REFP 3 C00115 BC00115
CALL JOB:SEARCH-R1
SET P0352 P0006
SFTON P0352
MOVL C00116 BC00116 V=166.7 PL=0
SFTOF
'------------------------
'W250A P
'------------------------
MOVJ C00117 BC00117 VJ=40.00
MOVL C00118 BC00118 V=166.7 PL=0
REFP 3 C00119 BC00119
CALL JOB:SEARCH-R1
SET P0353 P0006
SFTON P0353
MOVL C00120 BC00120 V=66.7 PL=0
REFP 3 C00121 BC00121
CALL JOB:SEARCH-R1
SET P0353 P0006
SFTON P0353
MOVL C00122 BC00122 V=66.7 PL=0
SFTOF
'------------------------
'W250A L
'------------------------
MOVJ C00123 BC00123 VJ=40.00
MOVL C00124 BC00124 V=166.7 PL=0
REFP 3 C00125 BC00125
CALL JOB:SEARCH-R1
SET P0354 P0006
SFTON P0354
MOVL C00126 BC00126 V=66.7 PL=0
REFP 3 C00127 BC00127
CALL JOB:SEARCH-R1
SET P0354 P0006
SFTON P0354
MOVL C00128 BC00128 V=166.7 PL=0
SFTOF
'------------------------
'W253A P
'------------------------
MOVJ C00129 BC00129 VJ=40.00
MOVL C00130 BC00130 V=166.7 PL=0
REFP 3 C00131 BC00131
CALL JOB:SEARCH-R1
SET P0355 P0006
SFTON P0355
MOVL C00132 BC00132 V=166.7 PL=0
REFP 3 C00133 BC00133
CALL JOB:SEARCH-R1
SET P0355 P0006
SFTON P0355
MOVL C00134 BC00134 V=166.7 PL=0
SFTOF
'------------------------
'W253A L
'------------------------
MOVJ C00135 BC00135 VJ=40.00
MOVL C00136 BC00136 V=166.7 PL=0
REFP 3 C00137 BC00137
CALL JOB:SEARCH-R1
SET P0356 P0006
SFTON P0356
MOVL C00138 BC00138 V=166.7 PL=0
REFP 3 C00139 BC00139
CALL JOB:SEARCH-R1
SET P0356 P0006
SFTON P0356
MOVL C00140 BC00140 V=166.7 PL=0
SFTOF
'------------------------
'W256A P
'------------------------
MOVJ C00141 BC00141 VJ=40.00
MOVL C00142 BC00142 V=166.7 PL=0
REFP 3 C00143 BC00143
CALL JOB:SEARCH-R1
SET P0357 P0006
SFTON P0357
MOVL C00144 BC00144 V=166.7 PL=0
REFP 3 C00145 BC00145
CALL JOB:SEARCH-R1
SET P0357 P0006
SFTON P0357
MOVL C00146 BC00146 V=166.7 PL=0
SFTOF
'------------------------
'W256A L
'------------------------
MOVJ C00147 BC00147 VJ=40.00
MOVL C00148 BC00148 V=166.7 PL=0
REFP 3 C00149 BC00149
CALL JOB:SEARCH-R1
SET P0358 P0006
SFTON P0358
MOVL C00150 BC00150 V=166.7 PL=0
REFP 3 C00151 BC00151
CALL JOB:SEARCH-R1
SET P0358 P0006
SFTON P0358
MOVL C00152 BC00152 V=166.7 PL=0
SFTOF
'------------------------
'W252A P
'------------------------
MOVL C00153 BC00153 V=666.7
MOVL C00154 BC00154 V=166.7 PL=0
REFP 3 C00155 BC00155
CALL JOB:SEARCH-R1
SET P0359 P0006
SFTON P0359
MOVL C00156 BC00156 V=166.7 PL=0
REFP 3 C00157 BC00157
CALL JOB:SEARCH-R1
SET P0359 P0006
SFTON P0359
MOVL C00158 BC00158 V=166.7 PL=0
SFTOF
'------------------------
'W252A L
'------------------------
MOVL C00159 BC00159 V=500.0
MOVL C00160 BC00160 V=166.7 PL=0
REFP 3 C00161 BC00161
CALL JOB:SEARCH-R1
SET P0360 P0006
SFTON P0360
MOVL C00162 BC00162 V=166.7 PL=0
REFP 3 C00163 BC00163
CALL JOB:SEARCH-R1
SET P0360 P0006
SFTON P0360
MOVL C00164 BC00164 V=166.7 PL=0
SFTOF
'------------------------
'W255A
'------------------------
MOVL C00165 BC00165 V=500.0
MOVL C00166 BC00166 V=166.7 PL=0
REFP 3 C00167 BC00167
CALL JOB:SEARCH-R1
SET P0361 P0006
SFTON P0361
MOVL C00168 BC00168 V=166.7 PL=0
REFP 3 C00169 BC00169
CALL JOB:SEARCH-R1
SET P0361 P0006
SFTON P0361
MOVL C00170 BC00170 V=166.7 PL=0
SFTOF
MOVL C00171 BC00171 V=666.7
MOVL C00172 BC00172 V=666.7
MOVL C00173 BC00173 V=666.7
MOVJ C00174 BC00174 VJ=40.00
MOVJ C00175 BC00175 VJ=40.00
COMM MOVJ C00176 BC00176 VJ=40.00
COMM MOVJ C00177 BC00177 VJ=40.00
COMM MOVJ C00178 BC00178 VJ=40.00
COMM MOVJ C00179 BC00179 VJ=40.00
COMM MOVJ C00180 BC00180 VJ=30.00
COMM '------------------------
COMM 'W61.3
COMM '------------------------
COMM MOVL C00181 BC00181 V=500.0
COMM MOVL C00182 BC00182 V=166.7 PL=0
COMM REFP 3 C00183 BC00183
COMM CALL JOB:SEARCH-R1
COMM SET P0400 P0006
COMM SFTON P0400
COMM MOVL C00184 BC00184 V=166.7 PL=0
COMM REFP 3 C00185 BC00185
COMM CALL JOB:SEARCH-R1
COMM SET P0400 P0006
COMM SFTON P0400
COMM MOVL C00186 BC00186 V=166.7 PL=0
COMM SFTOF
COMM 'BELKA PRZEJAZD
COMM MOVL C00187 BC00187 V=333.3
COMM '------------------------
COMM 'W61.5
COMM '------------------------
COMM MOVL C00188 BC00188 V=166.7 PL=0
COMM REFP 3 C00189 BC00189
COMM CALL JOB:SEARCH-R1
COMM SET P0401 P0006
COMM SFTON P0401
COMM MOVL C00190 BC00190 V=166.7 PL=0
COMM REFP 3 C00191 BC00191
COMM CALL JOB:SEARCH-R1
COMM SET P0401 P0006
COMM SFTON P0401
COMM MOVL C00192 BC00192 V=166.7 PL=0
COMM SFTOF
COMM '------------------------
COMM 'W61.7
COMM '------------------------
COMM MOVL C00193 BC00193 V=500.0
COMM MOVL C00194 BC00194 V=166.7 PL=0
COMM REFP 3 C00195 BC00195
COMM CALL JOB:SEARCH-R1
COMM SET P0402 P0006
COMM SFTON P0402
COMM MOVL C00196 BC00196 V=166.7 PL=0
COMM REFP 3 C00197 BC00197
COMM CALL JOB:SEARCH-R1
COMM SET P0402 P0006
COMM SFTON P0402
COMM MOVL C00198 BC00198 V=166.7 PL=0
COMM SFTOF
COMM MOVL C00199 BC00199 V=500.0
COMM '------------------------
COMM 'W61.10
COMM '------------------------
COMM MOVJ C00200 BC00200 VJ=30.00
COMM MOVJ C00201 BC00201 VJ=50.00
COMM MOVJ C00202 BC00202 VJ=50.00
COMM MOVL C00203 BC00203 V=500.0
COMM MOVL C00204 BC00204 V=166.7 PL=0
COMM REFP 3 C00205 BC00205
COMM CALL JOB:SEARCH-R1
COMM SET P0403 P0006
COMM SFTON P0403
COMM MOVL C00206 BC00206 V=166.7 PL=0
COMM REFP 3 C00207 BC00207
COMM CALL JOB:SEARCH-R1
COMM SET P0403 P0006
COMM SFTON P0403
COMM MOVL C00208 BC00208 V=166.7 PL=0
COMM SFTOF
COMM MOVL C00209 BC00209 V=333.3
COMM '------------------------
COMM 'W61.12
COMM '------------------------
COMM MOVL C00210 BC00210 V=666.7
COMM MOVL C00211 BC00211 V=166.7 PL=0
COMM REFP 3 C00212 BC00212
COMM CALL JOB:SEARCH-R1
COMM SET P0404 P0006
COMM SFTON P0404
COMM MOVL C00213 BC00213 V=166.7 PL=0
COMM REFP 3 C00214 BC00214
COMM CALL JOB:SEARCH-R1
COMM SET P0404 P0006
COMM SFTON P0404
COMM MOVL C00215 BC00215 V=166.7 PL=0
COMM SFTOF
COMM '------------------------
COMM 'W61.15
COMM '------------------------
COMM MOVL C00216 BC00216 V=666.7
COMM MOVL C00217 BC00217 V=166.7 PL=0
COMM REFP 3 C00218 BC00218
COMM CALL JOB:SEARCH-R1
COMM SET P0405 P0006
COMM SFTON P0405
COMM MOVL C00219 BC00219 V=166.7 PL=0
COMM REFP 3 C00220 BC00220
COMM CALL JOB:SEARCH-R1
COMM SET P0405 P0006
COMM SFTON P0405
COMM MOVL C00221 BC00221 V=166.7 PL=0
COMM SFTOF
COMM MOVL C00222 BC00222 V=666.7
COMM MOVJ C00223 BC00223 VJ=50.00
COMM MOVJ C00224 BC00224 VJ=50.00
COMM MOVJ C00225 BC00225 VJ=50.00
COMM '------------------------
COMM 'W61.17
COMM '------------------------
COMM MOVL C00226 BC00226 V=416.7
COMM MOVL C00227 BC00227 V=166.7 PL=0
COMM REFP 3 C00228 BC00228
COMM CALL JOB:SEARCH-R1
COMM SET P0406 P0006
COMM SFTON P0406
COMM MOVL C00229 BC00229 V=166.7 PL=0
COMM REFP 3 C00230 BC00230
COMM CALL JOB:SEARCH-R1
COMM SET P0406 P0006
COMM SFTON P0406
COMM MOVL C00231 BC00231 V=166.7 PL=0
COMM SFTOF
COMM MOVL C00232 BC00232 V=333.3
COMM '------------------------
COMM 'W61.20
COMM '------------------------
COMM MOVL C00233 BC00233 V=666.7
COMM MOVL C00234 BC00234 V=166.7 PL=0
COMM REFP 3 C00235 BC00235
COMM CALL JOB:SEARCH-R1
COMM SET P0407 P0006
COMM SFTON P0407
COMM MOVL C00236 BC00236 V=166.7 PL=0
COMM REFP 3 C00237 BC00237
COMM CALL JOB:SEARCH-R1
COMM SET P0407 P0006
COMM SFTON P0407
COMM MOVL C00238 BC00238 V=166.7 PL=0
COMM SFTOF
COMM '------------------------
COMM 'W61.23
COMM '------------------------
COMM MOVL C00239 BC00239 V=500.0
COMM MOVL C00240 BC00240 V=166.7 PL=0
COMM REFP 3 C00241 BC00241
COMM CALL JOB:SEARCH-R1
COMM SET P0408 P0006
COMM SFTON P0408
COMM MOVL C00242 BC00242 V=166.7 PL=0
COMM REFP 3 C00243 BC00243
COMM CALL JOB:SEARCH-R1
COMM SET P0408 P0006
COMM SFTON P0408
COMM MOVL C00244 BC00244 V=166.7 PL=0
COMM SFTOF
COMM MOVL C00245 BC00245 V=333.3
COMM MOVL C00246 BC00246 V=666.7
COMM MOVL C00247 BC00247 V=666.7
COMM '------------------------
COMM 'W61.25
COMM '------------------------
COMM MOVL C00248 BC00248 V=500.0
COMM MOVL C00249 BC00249 V=166.7 PL=0
COMM REFP 3 C00250 BC00250
COMM CALL JOB:SEARCH-R1
COMM SET P0409 P0006
COMM SFTON P0409
COMM MOVL C00251 BC00251 V=166.7 PL=0
COMM REFP 3 C00252 BC00252
COMM CALL JOB:SEARCH-R1
COMM SET P0409 P0006
COMM SFTON P0409
COMM MOVL C00253 BC00253 V=166.7 PL=0
COMM SFTOF
COMM MOVL C00254 BC00254 V=666.7
COMM MOVJ C00255 BC00255 VJ=50.00
COMM MOVJ C00256 BC00256 VJ=50.00
COMM GETE D040 P0409 (1)
COMM GETE D041 P0409 (2)
COMM GETE D042 P0409 (3)
COMM SETE P0410 (1) D040
COMM SETE P0410 (2) D041
COMM SETE P0410 (3) D042
COMM '------------------------
COMM 'W61.30
COMM '------------------------
COMM MOVL C00257 BC00257 V=500.0
COMM MOVL C00258 BC00258 V=166.7 PL=0
COMM REFP 3 C00259 BC00259
COMM CALL JOB:SEARCH-R1
COMM SET P0411 P0006
COMM SFTON P0411
COMM MOVL C00260 BC00260 V=166.7 PL=0
COMM REFP 3 C00261 BC00261
COMM CALL JOB:SEARCH-R1
COMM SET P0411 P0006
COMM SFTON P0411
COMM MOVL C00262 BC00262 V=166.7 PL=0
COMM SFTOF
COMM MOVL C00263 BC00263 V=666.7
COMM MOVJ C00264 BC00264 VJ=50.00
MOVJ C00265 BC00265 VJ=70.00
CALL JOB:FRONT_SEARCH_-90ST-2_5440
MOVJ C00266 BC00266 VJ=60.00
MOVJ C00267 BC00267 VJ=50.00
MOVJ C00268 BC00268 VJ=50.00
MOVL C00269 BC00269 V=666.7
MOVJ C00270 BC00270 VJ=30.00
'------------------------
'W65.3
'------------------------
SFTON P0300
MOVL C00271 BC00271 V=333.3
MOVL C00272 BC00272 V=166.7 PL=0
MACRO1 MJ#(0) ARGF10
ARCON
MOVL C00273 BC00273 V=10.8
ARCOF
MOVL C00274 BC00274 V=166.7
SFTOF
'------------------------
'W65.5
'------------------------
SFTON P0301
MOVL C00275 BC00275 V=666.7
MOVL C00276 BC00276 V=166.7 PL=0
MACRO1 MJ#(0) ARGF9
ARCON
MOVL C00277 BC00277 V=8.3
ARCOF
MOVL C00278 BC00278 V=166.7
SFTOF
MOVL C00279 BC00279 V=500.0
MOVL C00280 BC00280 V=666.7
MOVJ C00281 BC00281 VJ=40.00
COMM MOVJ C00282 BC00282 VJ=60.00
COMM '::::::::::::::::::::::::::::::::
COMM '::::::::::::::::::::::::::::::::
COMM '::::::::::::::::::::::::::::::::
COMM '::::::::::::::::::::::::::::::::
COMM '::::::::::::::::::::::::::::::::
COMM MOVJ C00283 BC00283 VJ=50.00
COMM MOVJ C00284 BC00284 VJ=50.00
COMM MOVJ C00285 BC00285 VJ=40.00
COMM MOVJ C00286 BC00286 VJ=40.00
COMM MOVJ C00287 BC00287 VJ=40.00
COMM MOVJ C00288 BC00288 VJ=40.00
COMM MOVL C00289 BC00289 V=666.7
COMM '------------------------
COMM 'W61.3
COMM '------------------------
COMM SFTON P0400
COMM ARCOF
COMM MOVL C00290 BC00290 V=500.0
COMM SFTOF
COMM 'BELKA PRZEJAZD
COMM '------------------------
COMM 'W61.5
COMM '------------------------
COMM SFTON P0401
COMM MOVL C00291 BC00291 V=666.7
COMM MOVL C00292 BC00292 V=166.7 PL=0
COMM MACRO1 MJ#(0) ARGF24
COMM ARCON
COMM MOVL C00293 BC00293 V=7.5
COMM ARCOF
COMM MOVL C00294 BC00294 V=250.0
COMM SFTOF
COMM MOVL C00295 BC00295 V=500.0
COMM MOVJ C00296 BC00296 VJ=40.00
COMM MOVJ C00297 BC00297 VJ=40.00
COMM MOVJ C00298 BC00298 VJ=50.00
COMM MOVJ C00299 BC00299 VJ=50.00
MOVJ C00300 BC00300 VJ=50.00
MOVJ C00301 BC00301 VJ=50.00
MOVL C00302 BC00302 V=666.7
'------------------------
'W250A
'------------------------
SFTON P0354
MOVL C00303 BC00303 V=666.7
MOVL C00304 BC00304 V=166.7 PL=0
MACRO1 MJ#(0) ARGF9
ARCON
SFTOF
SFTON P0353
MOVL C00305 BC00305 V=11.7
ARCOF
MOVL C00306 BC00306 V=333.3
SFTOF
MOVJ C00307 BC00307 VJ=50.00
MOVJ C00308 BC00308 VJ=60.00
MOVJ C00309 BC00309 VJ=40.00
MOVJ C00310 BC00310 VJ=50.00
MOVJ C00311 BC00311 VJ=40.00
MOVJ C00312 BC00312 VJ=30.00
MOVJ C00313 BC00313 VJ=15.00
'------------------------
'W65.7
'------------------------
SFTON P0302
MOVL C00314 BC00314 V=833.3
MOVL C00315 BC00315 V=166.7 PL=0
MACRO1 MJ#(0) ARGF10
ARCON
MOVL C00316 BC00316 V=10.8
ARCOF
MOVL C00317 BC00317 V=166.7
SFTOF
'------------------------
'W65.10
'------------------------
SFTON P0303
MOVL C00318 BC00318 V=666.7
MOVL C00319 BC00319 V=166.7 PL=0
ARCON
MOVL C00320 BC00320 V=10.8
ARCOF
MOVL C00321 BC00321 V=166.7
SFTOF
MOVL C00322 BC00322 V=333.3
MOVL C00323 BC00323 V=666.7
MOVJ C00324 BC00324 VJ=30.00
MOVJ C00325 BC00325 VJ=30.00
MOVJ C00326 BC00326 VJ=30.00
MOVJ C00327 BC00327 VJ=50.00
COMM '::::::::::::::::::::::::::::::::
COMM '::::::::::::::::::::::::::::::::
COMM '------------------------
COMM 'W61.7
COMM '------------------------
COMM '::::::::::::::::::::::::::::::::
COMM '::::::::::::::::::::::::::::::::
COMM MOVJ C00328 BC00328 VJ=30.00
COMM MOVJ C00329 BC00329 VJ=30.00
COMM MOVJ C00330 BC00330 VJ=40.00
COMM SFTON P0402
COMM MOVL C00331 BC00331 V=500.0
COMM MOVL C00332 BC00332 V=166.7 PL=0
COMM MACRO1 MJ#(0) ARGF24
COMM ARCON
COMM MOVL C00333 BC00333 V=7.5
COMM ARCOF
COMM MOVL C00334 BC00334 V=250.0
COMM SFTOF
COMM MOVJ C00335 BC00335 VJ=30.00
COMM MOVJ C00336 BC00336 VJ=40.00
COMM MOVJ C00337 BC00337 VJ=50.00
COMM '------------------------
COMM 'W61.10
COMM '------------------------
COMM SFTON P0403
COMM MOVL C00338 BC00338 V=500.0
COMM MOVL C00339 BC00339 V=166.7 PL=0
COMM MACRO1 MJ#(0) ARGF24
COMM ARCON
COMM MOVL C00340 BC00340 V=7.5
COMM ARCOF
COMM MOVL C00341 BC00341 V=250.0
COMM SFTOF
COMM MOVL C00342 BC00342 V=500.0
COMM MOVL C00343 BC00343 V=666.7
COMM MOVL C00344 BC00344 V=666.7
COMM MOVJ C00345 BC00345 VJ=50.00
COMM MOVJ C00346 BC00346 VJ=50.00
COMM MOVJ C00347 BC00347 VJ=50.00
COMM '::::::::::::::::::::::::
COMM '::::::::::::::::::::::::
COMM '::::::::::::::::::::::::
COMM '::::::::::::::::::::::::
COMM '::::::::::::::::::::::::
COMM '::::::::::::::::::::::::
COMM '::::::::::::::::::::::::
MOVJ C00348 BC00348 VJ=50.00
MOVJ C00349 BC00349 VJ=50.00
MOVJ C00350 BC00350 VJ=50.00
'------------------------
'W251B
'------------------------
MOVL C00351 BC00351 V=500.0
MOVL C00352 BC00352 V=500.0
SFTON P0350
MOVL C00353 BC00353 V=166.7 PL=0
MACRO1 MJ#(0) ARGF9
ARCON
SFTOF
SFTON P0349
MOVL C00354 BC00354 V=11.3
MOVL C00355 BC00355 V=11.3
ARCOF
MOVL C00356 BC00356 V=333.3
SFTOF
MOVJ C00357 BC00357 VJ=50.00
MOVJ C00358 BC00358 VJ=50.00
MOVJ C00359 BC00359 VJ=10.00
MOVJ C00360 BC00360 VJ=50.00
MOVJ C00361 BC00361 VJ=50.00
MOVJ C00362 BC00362 VJ=25.00
MOVJ C00363 BC00363 VJ=20.00
MOVJ C00364 BC00364 VJ=20.00
'------------------------
'W65.12
'------------------------
SFTON P0304
MOVL C00365 BC00365 V=333.3
MOVL C00366 BC00366 V=166.7 PL=0
MACRO1 MJ#(0) ARGF10
ARCON
MOVL C00367 BC00367 V=10.8
ARCOF
MOVL C00368 BC00368 V=166.7
SFTOF
'------------------------
'W65.15
'------------------------
SFTON P0305
MOVL C00369 BC00369 V=666.7
MOVL C00370 BC00370 V=166.7 PL=0
MACRO1 MJ#(0) ARGF9
ARCON
MOVL C00371 BC00371 V=10.8
ARCOF
MOVL C00372 BC00372 V=200.0
SFTOF
MOVL C00373 BC00373 V=250.0
MOVL C00374 BC00374 V=416.7
MOVL C00375 BC00375 V=666.7
COMM MOVJ C00376 BC00376 VJ=50.00
COMM MOVJ C00377 BC00377 VJ=50.00
COMM '::::::::::::::::::::::::
COMM '::::::::::::::::::::::::
COMM '::::::::::::::::::::::::
COMM '::::::::::::::::::::::::
COMM '::::::::::::::::::::::::
COMM '::::::::::::::::::::::::
COMM '::::::::::::::::::::::::
COMM MOVJ C00378 BC00378 VJ=50.00
COMM MOVJ C00379 BC00379 VJ=50.00
COMM MOVJ C00380 BC00380 VJ=50.00
COMM '::::::::::::::::::::::::::::::::
COMM '::::::::::::::::::::::::::::::::
COMM '------------------------
COMM 'W61.12
COMM '------------------------
COMM '::::::::::::::::::::::::::::::::
COMM '::::::::::::::::::::::::::::::::
COMM MOVL C00381 BC00381 V=833.3
COMM MOVL C00382 BC00382 V=666.7
COMM MOVL C00383 BC00383 V=500.0
COMM SFTON P0404
COMM MOVL C00384 BC00384 V=166.7 PL=0
COMM MACRO1 MJ#(0) ARGF24
COMM ARCON
COMM MOVL C00385 BC00385 V=6.7
COMM ARCOF
COMM MOVL C00386 BC00386 V=333.3
COMM SFTOF
COMM MOVL C00387 BC00387 V=500.0
COMM MOVL C00388 BC00388 V=666.7
COMM '------------------------
COMM 'W61.15
COMM '------------------------
COMM SFTON P0405
COMM MOVL C00389 BC00389 V=666.7
COMM MOVL C00390 BC00390 V=166.7 PL=0
COMM MACRO1 MJ#(0) ARGF24
COMM ARCON
COMM MOVL C00391 BC00391 V=6.7
COMM ARCOF
COMM MOVL C00392 BC00392 V=250.0
COMM SFTOF
COMM MOVJ C00393 BC00393 VJ=40.00
COMM MOVJ C00394 BC00394 VJ=40.00
COMM MOVJ C00395 BC00395 VJ=40.00
COMM MOVJ C00396 BC00396 VJ=40.00
COMM '::::::::::::::::::::::::
COMM '::::::::::::::::::::::::
COMM '::::::::::::::::::::::::
COMM '::::::::::::::::::::::::
COMM '::::::::::::::::::::::::
COMM '::::::::::::::::::::::::
COMM '::::::::::::::::::::::::
COMM MOVJ C00397 BC00397 VJ=40.00
COMM MOVJ C00398 BC00398 VJ=40.00
COMM '------------------------
COMM 'W252B
COMM '------------------------
SFTON P0359
MOVL C00399 BC00399 V=666.7
MOVL C00400 BC00400 V=166.7 PL=0
MACRO1 MJ#(0) ARGF9
ARCON
SFTOF
SFTON P0358
MOVL C00401 BC00401 V=10.8
ARCOF
MOVL C00402 BC00402 V=250.0
SFTOF
MOVJ C00403 BC00403 VJ=50.00
MOVJ C00404 BC00404 VJ=50.00
MOVJ C00405 BC00405 VJ=60.00
MOVJ C00406 BC00406 VJ=40.00
MOVJ C00407 BC00407 VJ=30.00
MOVL C00408 BC00408 V=500.0
MOVL C00409 BC00409 V=333.3
'------------------------
'W65.17
'------------------------
SFTON P0306
MOVL C00410 BC00410 V=333.3
MOVL C00411 BC00411 V=166.7 PL=0
MACRO1 MJ#(0) ARGF10
ARCON
MOVL C00412 BC00412 V=10.8
ARCOF
MOVL C00413 BC00413 V=166.7
SFTOF
MOVL C00414 BC00414 V=333.3
MOVL C00415 BC00415 V=500.0
MOVL C00416 BC00416 V=500.0
MOVJ C00417 BC00417 VJ=40.00
COMM MOVJ C00418 BC00418 VJ=60.00
COMM MOVJ C00419 BC00419 VJ=60.00
COMM '::::::::::::::::::::::::
COMM '::::::::::::::::::::::::
COMM '::::::::::::::::::::::::
COMM '::::::::::::::::::::::::
COMM '::::::::::::::::::::::::
COMM '::::::::::::::::::::::::
COMM '::::::::::::::::::::::::
COMM MOVJ C00420 BC00420 VJ=60.00
COMM '::::::::::::::::::::::::::::::::
COMM '::::::::::::::::::::::::::::::::
COMM '------------------------
COMM 'W61.17
COMM '------------------------
COMM '::::::::::::::::::::::::::::::::
COMM '::::::::::::::::::::::::::::::::
COMM SFTON P0406
COMM MOVJ C00421 BC00421 VJ=40.00
COMM MOVL C00422 BC00422 V=500.0
COMM MOVL C00423 BC00423 V=166.7 PL=0
COMM MACRO1 MJ#(0) ARGF24
COMM ARCON
COMM MOVL C00424 BC00424 V=6.7
COMM ARCOF
COMM MOVL C00425 BC00425 V=333.3
COMM SFTOF
COMM MOVJ C00426 BC00426 VJ=30.00
COMM MOVJ C00427 BC00427 VJ=40.00
COMM MOVJ C00428 BC00428 VJ=50.00
COMM '------------------------
COMM 'W253A
'------------------------
COMM MOVJ C00429 BC00429 VJ=50.00
MOVJ C00430 BC00430 VJ=50.00
SFTON P0356
MOVL C00431 BC00431 V=500.0
MOVL C00432 BC00432 V=500.0
MOVL C00433 BC00433 V=166.7 PL=0
MACRO1 MJ#(0) ARGF9
ARCON
SFTOF
SFTON P0355
MOVL C00434 BC00434 V=11.3
ARCOF
MOVL C00435 BC00435 V=333.3
SFTOF
MOVJ C00436 BC00436 VJ=50.00
'------------------------
'W65.20
'------------------------
COMM MOVJ C00437 BC00437 VJ=50.00
COMM MOVJ C00438 BC00438 VJ=50.00
COMM MOVJ C00439 BC00439 VJ=50.00
COMM '::::::::::::::::::::::::
COMM '::::::::::::::::::::::::
COMM '::::::::::::::::::::::::
COMM '::::::::::::::::::::::::
COMM '::::::::::::::::::::::::
COMM '::::::::::::::::::::::::
COMM '::::::::::::::::::::::::
COMM MOVJ C00440 BC00440 VJ=40.00
COMM MOVJ C00441 BC00441 VJ=40.00
COMM '::::::::::::::::::::::::::::::::
COMM '::::::::::::::::::::::::::::::::
COMM '------------------------
COMM 'W61.20
COMM '------------------------
COMM '::::::::::::::::::::::::::::::::
COMM '::::::::::::::::::::::::::::::::
COMM SFTON P0407
COMM MOVL C00442 BC00442 V=666.7
COMM MOVL C00443 BC00443 V=333.3
COMM MOVL C00444 BC00444 V=166.7 PL=0
COMM MACRO1 MJ#(0) ARGF24
COMM ARCON
COMM MOVL C00445 BC00445 V=6.7
COMM ARCOF
COMM MOVL C00446 BC00446 V=250.0
COMM SFTOF
COMM '::::::::::::::::::::::::
COMM '::::::::::::::::::::::::
COMM '::::::::::::::::::::::::
COMM '::::::::::::::::::::::::
COMM '::::::::::::::::::::::::
COMM MOVL C00447 BC00447 V=500.0
COMM MOVJ C00448 BC00448 VJ=50.00
COMM MOVJ C00449 BC00449 VJ=50.00
COMM MOVJ C00450 BC00450 VJ=50.00
COMM '------------------------
COMM 'W254A
COMM '------------------------
COMM MOVJ C00451 BC00451 VJ=50.00
MOVJ C00452 BC00452 VJ=50.00
SFTON P0352
MOVL C00453 BC00453 V=666.7
MOVL C00454 BC00454 V=500.0
MOVL C00455 BC00455 V=250.0 PL=0
MACRO1 MJ#(0) ARGF9
ARCON
SFTOF
SFTON P0351
MOVL C00456 BC00456 V=11.2
ARCOF
MOVL C00457 BC00457 V=333.3
MOVL C00458 BC00458 V=666.7
SFTOF
COMM MOVJ C00459 BC00459 VJ=50.00
COMM MOVJ C00460 BC00460 VJ=80.00
COMM MOVJ C00461 BC00461 VJ=50.00
MOVJ C00462 BC00462 VJ=50.00
MOVJ C00463 BC00463 VJ=30.00
MOVL C00464 BC00464 V=666.7
'------------------------
'W65.23
'------------------------
SFTON P0308
MOVL C00465 BC00465 V=333.3
MOVL C00466 BC00466 V=166.7
MOVL C00467 BC00467 V=166.7 PL=0
MACRO1 MJ#(0) ARGF10
ARCON
MOVL C00468 BC00468 V=10.8
ARCOF
MOVL C00469 BC00469 V=250.0
SFTOF
'------------------------
'W65.25
'------------------------
SFTON P0309
MOVL C00470 BC00470 V=666.7
MOVL C00471 BC00471 V=166.7
MOVL C00472 BC00472 V=166.7 PL=0
ARCON
MOVL C00473 BC00473 V=10.8
ARCOF
MOVL C00474 BC00474 V=250.0
SFTOF
MOVL C00475 BC00475 V=250.0
MOVL C00476 BC00476 V=500.0
MOVL C00477 BC00477 V=666.7
MOVL C00478 BC00478 V=666.7
MOVJ C00479 BC00479 VJ=40.00
MOVJ C00480 BC00480 VJ=40.00
MOVJ C00481 BC00481 VJ=50.00
COMM '::::::::::::::::::::::::
COMM '::::::::::::::::::::::::
COMM '::::::::::::::::::::::::
COMM '::::::::::::::::::::::::
COMM '::::::::::::::::::::::::
COMM '::::::::::::::::::::::::
COMM '::::::::::::::::::::::::
COMM MOVJ C00482 BC00482 VJ=50.00
COMM MOVJ C00483 BC00483 VJ=50.00
COMM MOVJ C00484 BC00484 VJ=50.00
COMM '::::::::::::::::::::::::::::::::
COMM '::::::::::::::::::::::::::::::::
COMM '------------------------
COMM 'W61.23
COMM '------------------------
COMM '::::::::::::::::::::::::::::::::
COMM '::::::::::::::::::::::::::::::::
COMM SFTON P0408
COMM MOVL C00485 BC00485 V=500.0
COMM MOVL C00486 BC00486 V=666.7
COMM MOVL C00487 BC00487 V=166.7 PL=0
COMM MACRO1 MJ#(0) ARGF24
COMM ARCON
COMM MOVL C00488 BC00488 V=8.3
COMM ARCOF
COMM MOVL C00489 BC00489 V=250.0
COMM SFTOF
COMM MOVL C00490 BC00490 V=666.7
COMM '------------------------
COMM 'W61.25
COMM '------------------------
COMM SFTON P0409
COMM MOVL C00491 BC00491 V=500.0
COMM MOVL C00492 BC00492 V=166.7 PL=0
COMM MACRO1 MJ#(0) ARGF24
COMM ARCON
COMM MOVL C00493 BC00493 V=8.3
COMM ARCOF
COMM MOVL C00494 BC00494 V=166.7
COMM SFTOF
COMM MOVL C00495 BC00495 V=500.0
COMM MOVJ C00496 BC00496 VJ=20.00
COMM '::::::::::::::::::::::::
COMM '::::::::::::::::::::::::
COMM '::::::::::::::::::::::::
COMM '::::::::::::::::::::::::
COMM '::::::::::::::::::::::::
COMM MOVJ C00497 BC00497 VJ=50.00
COMM MOVJ C00498 BC00498 VJ=50.00
MOVJ C00499 BC00499 VJ=40.00
'------------------------
'W255A
MOVL C00500 BC00500 V=500.0
MOVL C00501 BC00501 V=666.7
SFTON P0361
MOVL C00502 BC00502 V=166.7 PL=0
MACRO1 MJ#(0) ARGF9
ARCON
MOVL C00503 BC00503 V=11.2
MOVL C00504 BC00504 V=10.8
ARCOF
MOVL C00505 BC00505 V=333.3
SFTOF
MOVL C00506 BC00506 V=666.7
MOVL C00507 BC00507 V=666.7
MOVL C00508 BC00508 V=666.7
MOVJ C00509 BC00509 VJ=50.00
MOVJ C00510 BC00510 VJ=70.00
MOVJ C00511 BC00511 VJ=70.00
MOVJ C00512 BC00512 VJ=50.00
MOVJ C00513 BC00513 VJ=50.00
MOVJ C00514 BC00514 VJ=50.00
MOVL C00515 BC00515 V=500.0
'------------------------
'W31.28
'------------------------
MOVL C00516 BC00516 V=333.3
MOVL C00517 BC00517 V=333.3
MACRO1 MJ#(0) ARGF10
SFTON P0311
MOVL C00518 BC00518 V=166.7
ARCON
MOVL C00519 BC00519 V=10.8
ARCOF
MOVL C00520 BC00520 V=250.0
MOVL C00521 BC00521 V=250.0
MOVL C00522 BC00522 V=200.0
ARCON
MOVL C00523 BC00523 V=10.8
ARCOF
MOVL C00524 BC00524 V=166.7
MOVL C00525 BC00525 V=333.3
SFTOF
SFTON P0312
MOVL C00526 BC00526 V=166.7
ARCON
MOVL C00527 BC00527 V=10.8
ARCOF
MOVL C00528 BC00528 V=166.7
MOVL C00529 BC00529 V=166.7
MOVL C00530 BC00530 V=166.7
ARCON
MOVL C00531 BC00531 V=10.8
ARCOF
'------------------------
SFTOF
MOVL C00532 BC00532 V=250.0
MOVL C00533 BC00533 V=416.7
MOVL C00534 BC00534 V=500.0
MOVL C00535 BC00535 V=500.0
MOVL C00536 BC00536 V=666.7
MOVJ C00537 BC00537 VJ=25.00
COMM '::::::::::::::::::::::::
COMM '::::::::::::::::::::::::
COMM '::::::::::::::::::::::::
COMM '::::::::::::::::::::::::
COMM '::::::::::::::::::::::::
COMM '::::::::::::::::::::::::
COMM '::::::::::::::::::::::::
COMM MOVJ C00538 BC00538 VJ=20.00
COMM MOVJ C00539 BC00539 VJ=30.00
COMM '::::::::::::::::::::::::::::::::
COMM '::::::::::::::::::::::::::::::::
COMM '------------------------
COMM 'W61.30
COMM '------------------------
COMM '::::::::::::::::::::::::::::::::
COMM '::::::::::::::::::::::::::::::::
COMM SFTON P0411
COMM MOVL C00540 BC00540 V=500.0
COMM MOVL C00541 BC00541 V=166.7 PL=0
COMM MACRO1 MJ#(0) ARGF24
COMM ARCON
COMM MOVL C00542 BC00542 V=7.5
COMM ARCOF
COMM MOVL C00543 BC00543 V=250.0
COMM MOVL C00544 BC00544 V=500.0
COMM MOVL C00545 BC00545 V=166.7 PL=0
COMM MACRO1 MJ#(0) ARGF24
COMM ARCON
COMM MOVL C00546 BC00546 V=7.5
COMM ARCOF
COMM MOVL C00547 BC00547 V=250.0
COMM SFTOF
COMM MOVL C00548 BC00548 V=500.0
COMM SFTOF
COMM MOVL C00549 BC00549 V=500.0
COMM MOVJ C00550 BC00550 VJ=25.00
MOVJ C00551 BC00551 VJ=50.00
MOVJ C00552 BC00552 VJ=50.00
MOVJ C00553 BC00553 VJ=60.00
'------------------------
'W256A
'------------------------
MOVJ C00554 BC00554 VJ=60.00
MOVJ C00555 BC00555 VJ=60.00
SFTON P0358
MOVL C00556 BC00556 V=666.7
MOVL C00557 BC00557 V=250.0
MOVL C00558 BC00558 V=166.7 PL=0
MACRO1 MJ#(0) ARGF9
ARCON
SFTOF
SFTON P0357
MOVL C00559 BC00559 V=11.2
ARCOF
MOVL C00560 BC00560 V=333.3
SFTOF
MOVJ C00561 BC00561 VJ=50.00
MOVJ C00562 BC00562 VJ=50.00
CALL JOB:FRONT_WELD_-90ST-2_5440
CALL JOB:MOVE_OUT_OF_TUNNEL
END
